ABB RobotStudio station: PaletizadoTPL2.rsstn

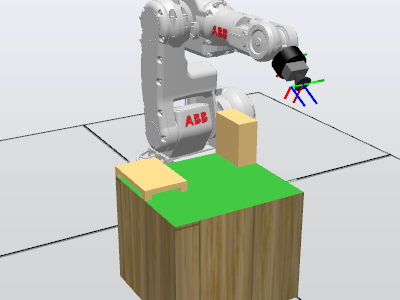
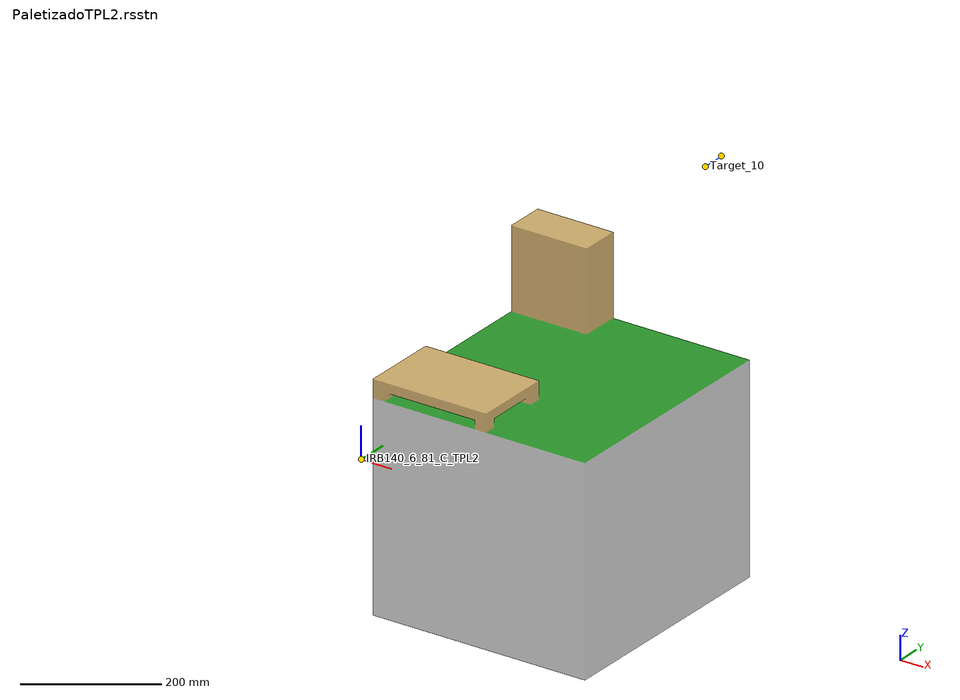
[picture v1: parts stored in the station drawn from their meshes, with robot base, taught points and paths (robot models come from the ABB library and are not in the file)]
Station Paletizado (saved by RobotStudio 25.5.11605.0)
Controller IRB140_6_81_TPL2
  mechanical unit ROB_1: IRB140_6_81_C_TPL2, 6 joints, base frame (0, 0, 0) mm
Layout (positions relative to the parent item):
  - Mesa [part], size 365 x 405 x 340 mm
  - Pallet [part], size 195 x 130 x 30 mm
  - Pieza1 [part], size 130 x 65 x 15 mm
  - Pieza2 [part], size 130 x 65 x 15 mm
  - Pieza3 [part], size 130 x 65 x 15 mm
  - Pieza4 [part], size 130 x 65 x 15 mm
  - Pieza5 [part], size 130 x 65 x 15 mm
  - Pieza6 [part], size 130 x 65 x 15 mm
  - Pieza7 [part], size 130 x 65 x 15 mm
  - Pieza8 [part], size 130 x 65 x 15 mm
  - Pieza9 [part], size 130 x 65 x 15 mm
  - Sopapa [mechanism] at (506.29, 39.79, 679.5) mm, rotated rx 180 ry 60 rz 180 deg
      TCP Sopapa at (0, -5, 103) mm
      links: Sopapa
  - IRB140_6_81_C_TPL2 [mechanism, from %ABB.RobotStudio.Models.IRB140%\IRB140_6_81_C_G_03.rslib] at (0, 0, 0) mm; joint values [0.0882, 0.0049, -0.0049, -0.1514, 0.5303, 0.175] (rad or m)
Attachment: Sopapa is attached to IRB140_6_81_C_TPL2 / Link6
EventTableEntry 1212: Group=, Trigger=DO_Pinza 1213, Actions=[EventTableActionAttach 1214], Comment=, ActivationMode=2, Cyclic=false
EventTableTriggerIO 1213: IOValue=[1], IRC5Controller=? -1, Operator=0, SignalSource=? -1
EventTableActionAttach 1214: AttachmentParent=Sopapa 1252, AttachmentChild=? -1, MountObject=false, Offset=[X=1, Y=0, Z=0, W=0, X=0, Y=1, Z=0, W=0, X=0, Y=0, Z=1, W=0, X=0, Y=0, Z=0, W=1], FlangeIndext=0, FindNearest=true
EventTableEntry 1219: Group=, Trigger=DO_Pinza 1220, Actions=[EventTableActionDetach 1221], Comment=, ActivationMode=2, Cyclic=false
EventTableTriggerIO 1220: IOValue=[0], IRC5Controller=? -1, Operator=0, SignalSource=? -1
EventTableActionDetach 1221: AttachmentParent=Sopapa 1252, AttachmentChild=? -1
Targets, tools, work objects and paths stored in the station, written as RAPID:
! task T_ROB1
MODULE Module1
  PERS tooldata Sopapa:=[TRUE,[[0,-5,103],[1,0,0,0]],[0.5,[0,0,40],[1,0,0,0],0,0,0]];
  CONST robtarget Target_10:=[[595.492267836,-5,628],[0.5,0,0.866025404,0],[0,0,0,0],[9E+09,9E+09,9E+09,9E+09,9E+09,9E+09]];
  CONST robtarget Target_20:=[[595.492192643,34.78927249,628.000011052],[0.500000018,0.000000003,0.866025394,0.000000005],[0,-1,0,0],[9E+09,9E+09,9E+09,9E+09,9E+09,9E+09]];
  PROC main()
    Path_10;
  ENDPROC
  PROC Path_10()
    MoveL Target_10,v1000,z100,Sopapa\WObj:=wobj0;
    MoveL Target_20,v1000,z100,Sopapa\WObj:=wobj0;
  ENDPROC
ENDMODULE

